/// Saturation. Limits the value to a minimum and maximum value
FUNCTION FUN_SaturationPointer_UInt : REAL
VAR_INPUT
	pValue			:POINTER TO UINT;	// Value				
	fMin			:REAL;				// Saturation min value
	fMax			:REAL;				// Saturation max value
END_VAR
VAR_OUTPUT
	bSaturation		:BOOL;
END_VAR

bSaturation := FALSE;
IF UINT_TO_REAL(pValue^) < fMin THEN
	pValue^ := REAL_TO_UINT(fMin);
	bSaturation := TRUE;
ELSIF UINT_TO_REAL(pValue^) > fMax THEN
	pValue^ := REAL_TO_UINT(fMax);
	bSaturation := TRUE;
END_IF

END_FUNCTION

(* stored: Version 1.1.0.1, ProductVersion 3.1.4024.12
   POU FUN_SaturationPointer_UInt: Id {62b11368-6aa0-4488-b43e-dfeb6ed836da}, SpecialFunc None *)
